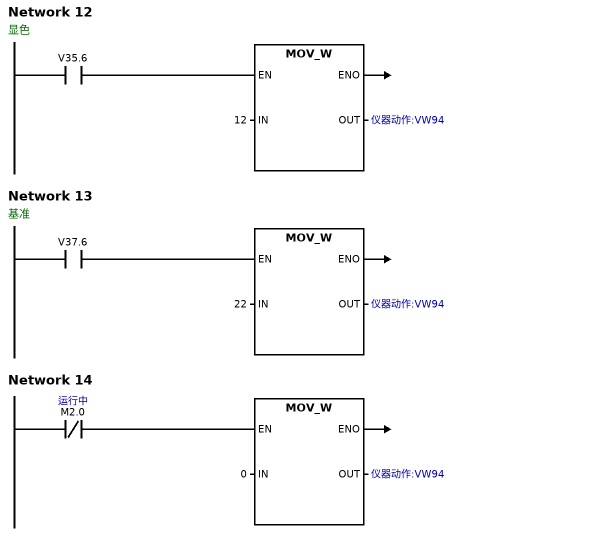
[picture p96: SBR35 networks 12-14]
Network 12
// 显色
LD     V35.6
MOVW   12, 仪器动作:VW94
Network 13
// 基准
LD     V37.6
MOVW   22, 仪器动作:VW94
Network 14
LDN    运行中:M2.0
MOVW   0, 仪器动作:VW94
END_SUBROUTINE_BLOCK

SUBROUTINE_BLOCK 三层:SBR36
TITLE=子程序注释
BEGIN
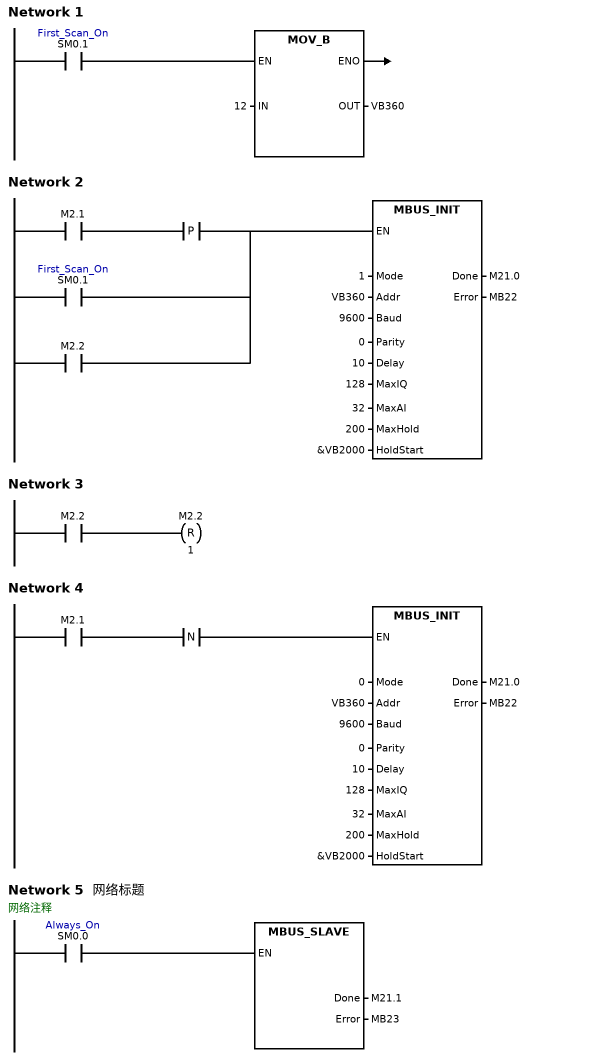
Network 1
LD     First_Scan_On:SM0.1
MOVB   12, VB360
Network 2
LD     M2.1
EU
O      First_Scan_On:SM0.1
O      M2.2
CALL   MBUS_INIT:SBR30, 1, VB360, 9600, 0, 10, 128, 32, 200, &VB2000, M21.0, MB22
Network 3
LD     M2.2
R      M2.2, 1
Network 4
LD     M2.1
ED
CALL   MBUS_INIT:SBR30, 0, VB360, 9600, 0, 10, 128, 32, 200, &VB2000, M21.0, MB22
Network 5 // 网络标题
// 网络注释
LD     Always_On:SM0.0
CALL   MBUS_SLAVE:SBR31, M21.1, MB23
END_SUBROUTINE_BLOCK

SUBROUTINE_BLOCK 计算A:SBR37
TITLE=
VAR_INPUT
显色1:REAL;	// LD0 
基准1:REAL;	// LD4 
END_VAR
VAR_OUTPUT
A1:REAL;	// LD8 
END_VAR
BEGIN
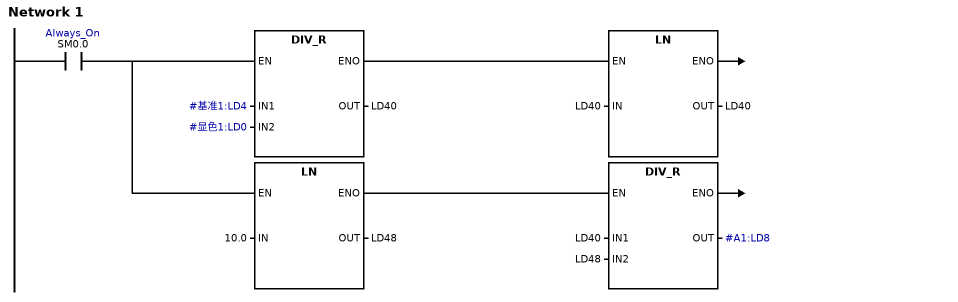
Network 1
LD     Always_On:SM0.0
LPS
MOVR   #基准1:LD4, LD40
AENO
/R     #显色1:LD0, LD40
AENO
LN     LD40, LD40
LPP
LN     10.0, LD48
AENO
MOVR   LD40, #A1:LD8
/R     LD48, #A1:LD8
Network 2 // 网络标题
// 网络注释
END_SUBROUTINE_BLOCK

SUBROUTINE_BLOCK 动态管控反控:SBR38
TITLE=子程序注释
BEGIN
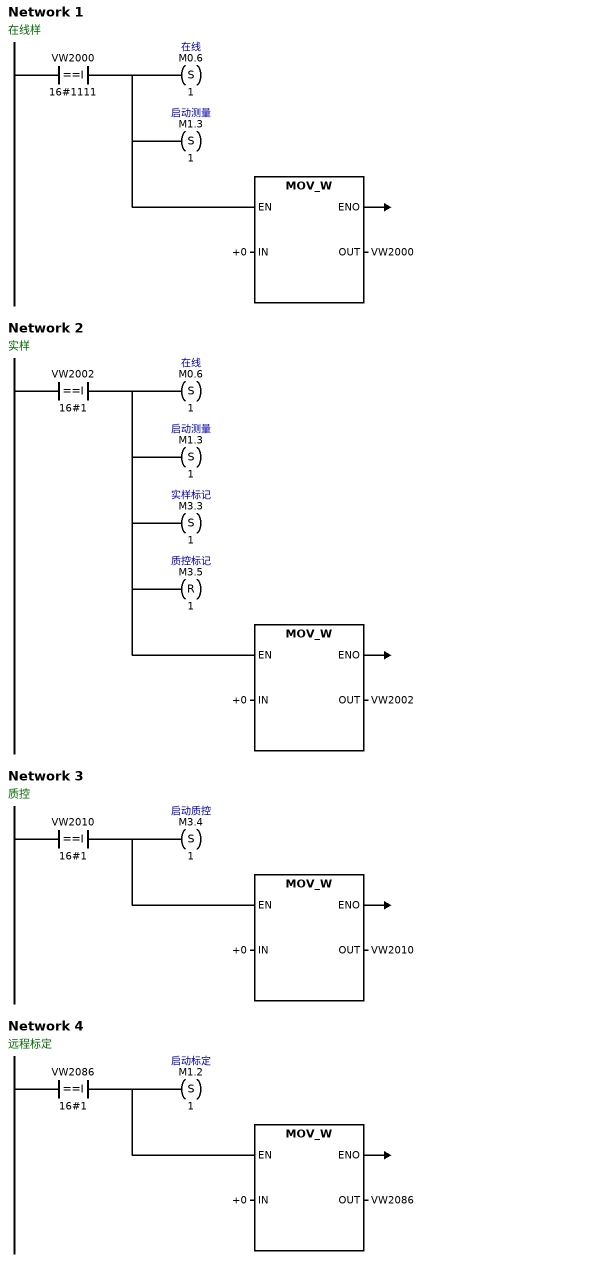
Network 1
// 在线样
LDW=   VW2000, 16#1111
S      在线:M0.6, 1
S      启动测量:M1.3, 1
MOVW   +0, VW2000
Network 2
// 实样
LDW=   VW2002, 16#1
S      在线:M0.6, 1
S      启动测量:M1.3, 1
S      实样标记:M3.3, 1
R      质控标记:M3.5, 1
MOVW   +0, VW2002
Network 3
// 质控
LDW=   VW2010, 16#1
S      启动质控:M3.4, 1
MOVW   +0, VW2010
Network 4
// 远程标定
LDW=   VW2086, 16#1
S      启动标定:M1.2, 1
MOVW   +0, VW2086
Network 5 // 网络标题
// 网络注释
END_SUBROUTINE_BLOCK

SUBROUTINE_BLOCK 填充:SBR39
TITLE=子程序注释
BEGIN
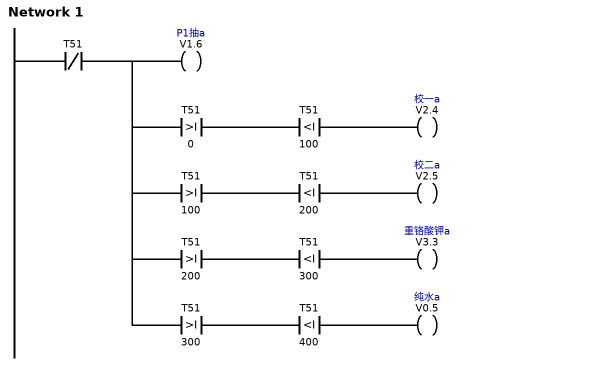
Network 1
LDN    T51
LPS
=      P1抽a:V1.6
AW>    T51, 0
AW<    T51, 100
=      校一a:V2.4
LRD
AW>    T51, 100
AW<    T51, 200
=      校二a:V2.5
LRD
AW>    T51, 200
AW<    T51, 300
=      重铬酸钾a:V3.3
LPP
AW>    T51, 300
AW<    T51, 400
=      纯水a:V0.5
Network 2 // 网络标题
// 网络注释
END_SUBROUTINE_BLOCK

SUBROUTINE_BLOCK 一键清洗:SBR40
TITLE=子程序注释
BEGIN
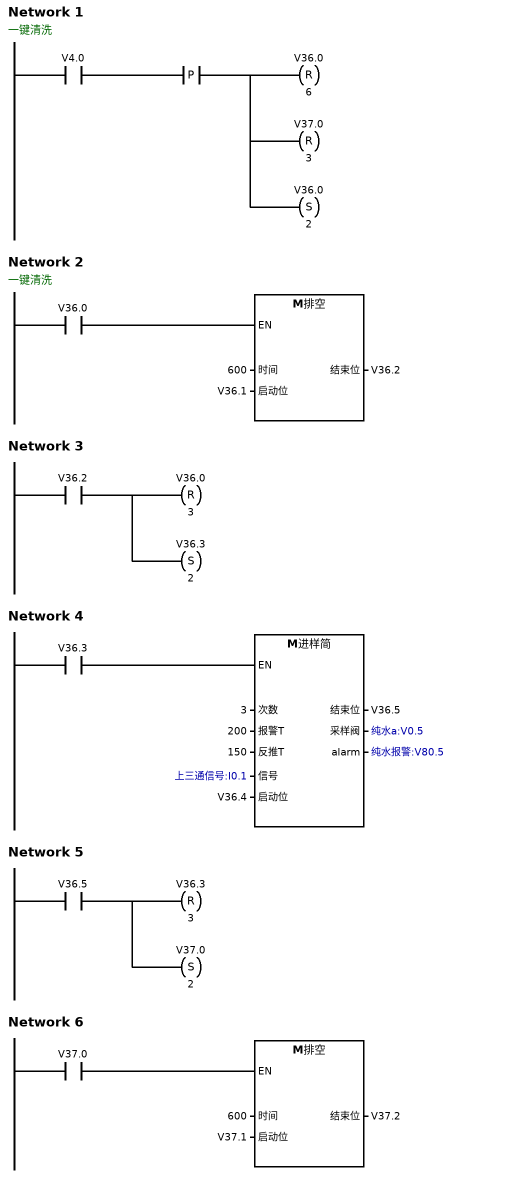
Network 1
// 一键清洗
LD     V4.0
EU
R      V36.0, 6
R      V37.0, 3
S      V36.0, 2
Network 2
// 一键清洗
LD     V36.0
CALL   M排空:SBR5, 600, V36.1, V36.2
Network 3
LD     V36.2
R      V36.0, 3
S      V36.3, 2
Network 4
LD     V36.3
CALL   M进样简:SBR1, 3, 200, 150, 上三通信号:I0.1, V36.4, V36.5, 纯水a:V0.5, 纯水报警:V80.5
Network 5
LD     V36.5
R      V36.3, 3
S      V37.0, 2
Network 6
LD     V37.0
CALL   M排空:SBR5, 600, V37.1, V37.2
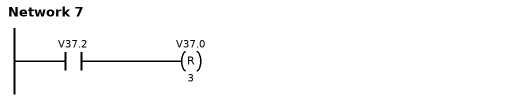
Network 7
LD     V37.2
R      V37.0, 3
Network 8 // 网络标题
// 网络注释
END_SUBROUTINE_BLOCK

SUBROUTINE_BLOCK 计算KB:SBR41
TITLE=
VAR_INPUT
A1:REAL;	// LD0 
浓度1:REAL;	// LD4 
A2:REAL;	// LD8 
浓度2:REAL;	// LD12 
END_VAR
VAR_OUTPUT
K:REAL;	// LD16 
b:REAL;	// LD20 
END_VAR
BEGIN
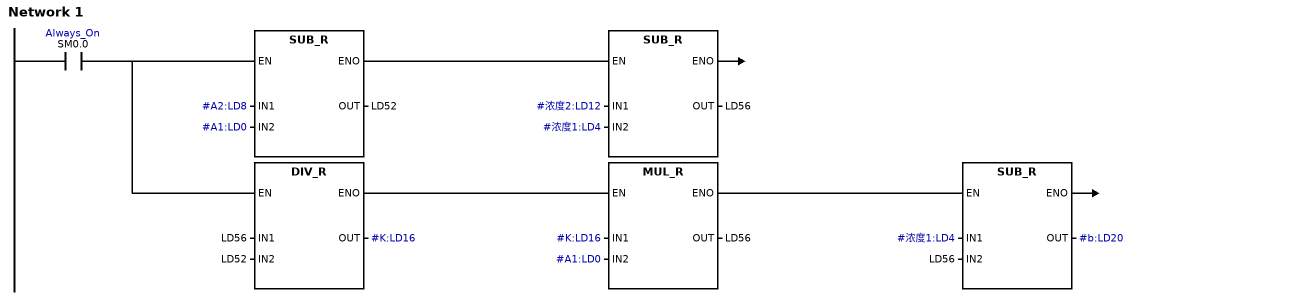
Network 1
LD     Always_On:SM0.0
LPS
MOVR   #A2:LD8, LD52
AENO
-R     #A1:LD0, LD52
AENO
MOVR   #浓度2:LD12, LD56
-R     #浓度1:LD4, LD56
LPP
MOVR   LD56, #K:LD16
AENO
/R     LD52, #K:LD16
AENO
MOVR   #K:LD16, LD56
AENO
*R     #A1:LD0, LD56
AENO
MOVR   #浓度1:LD4, #b:LD20
-R     LD56, #b:LD20
Network 2 // 网络标题
// 网络注释
END_SUBROUTINE_BLOCK

DATA_BLOCK_TAB 用户定义1
BEGIN
         操作密码, 888
         管理密码, 999
         超级密码, 8989
VD664    0.15                //重铬酸钾
VW332    2000                //默认量程
END_DATA_BLOCK_TAB
